# EPICS substitutions: apps/sensorProbeApp/Db/hallWeather.substitutions
file "db/sensorProbe_temperature.db" {
  pattern { P, A, C, HOST }
  { "B_HW_AKCP2", "B_SYS_WEATHER_FC_L1", "1", "%(AKCP2)" }
  { "B_HW_AKCP2", "B_SYS_WEATHER_FC_L2", "2", "%(AKCP2)" }
  { "B_HW_AKCP2", "B_SYS_WEATHER_FC_L3", "3", "%(AKCP2)" }
  { "B_HW_AKCP1", "B_SYS_WEATHER_SF_L1", "0", "%(AKCP1)" }
  { "B_HW_AKCP1", "B_SYS_WEATHER_SW",    "1", "%(AKCP1)" }
  { "B_HW_AKCP3", "B_SYS_WEATHER_PT",    "0", "%(AKCP3)" }
  { "B_HW_AKCP5", "B_SYS_WEATHER_CH",    "0", "%(AKCP5)" }
  { "B_HW_AKCP4", "B_SYS_WEATHER_CH_L",  "0", "%(AKCP4)" }
  { "B_HW_AKCP4", "B_SYS_WEATHER_CH_R",  "3", "%(AKCP4)" }
}
file "db/sensorProbe_humidity.db" {
  pattern { P, A, C, HOST }
  { "B_HW_AKCP2", "B_SYS_WEATHER_FC_L1", "1", "%(AKCP2)" }
  { "B_HW_AKCP2", "B_SYS_WEATHER_FC_L2", "2", "%(AKCP2)" }
  { "B_HW_AKCP2", "B_SYS_WEATHER_FC_L3", "3", "%(AKCP2)" }
  { "B_HW_AKCP1", "B_SYS_WEATHER_SF_L1", "0", "%(AKCP1)" }
  { "B_HW_AKCP1", "B_SYS_WEATHER_SW",    "1", "%(AKCP1)" }
  { "B_HW_AKCP3", "B_SYS_WEATHER_PT",    "0", "%(AKCP3)" }
  { "B_HW_AKCP5", "B_SYS_WEATHER_CH",    "0", "%(AKCP5)" }
  { "B_HW_AKCP4", "B_SYS_WEATHER_CH_L",  "0", "%(AKCP4)" }
  { "B_HW_AKCP4", "B_SYS_WEATHER_CH_R",  "3", "%(AKCP4)" }
}
